# EPICS substitutions: ospreyEVRSup/Db/ospreyEVR.substitutions
#   Undefined macros
#
# P - Common record name prefix
# NAME - Device instance name

file "perEVR.template" {
pattern { P,  NAME }
  { "\$(P)", "\$(NAME)" }
}

file "perEVRhwTrigger.template" {
pattern { P,     NAME   ,  I }
  { "\$(P)", "\$(NAME)", "1" }
  { "\$(P)", "\$(NAME)", "2" }
  { "\$(P)", "\$(NAME)", "3" }
  { "\$(P)", "\$(NAME)", "4" }
}

file "perEVRevent.template" {
pattern { P,     NAME,     E }
  { "\$(P)", "\$(NAME)", "001" }
  { "\$(P)", "\$(NAME)", "002" }
  { "\$(P)", "\$(NAME)", "003" }
  { "\$(P)", "\$(NAME)", "004" }
  { "\$(P)", "\$(NAME)", "005" }
  { "\$(P)", "\$(NAME)", "006" }
  { "\$(P)", "\$(NAME)", "007" }
  { "\$(P)", "\$(NAME)", "008" }
  { "\$(P)", "\$(NAME)", "009" }
  { "\$(P)", "\$(NAME)", "010" }
  { "\$(P)", "\$(NAME)", "011" }
  { "\$(P)", "\$(NAME)", "012" }
  { "\$(P)", "\$(NAME)", "013" }
  { "\$(P)", "\$(NAME)", "014" }
  { "\$(P)", "\$(NAME)", "015" }
  { "\$(P)", "\$(NAME)", "016" }
  { "\$(P)", "\$(NAME)", "017" }
  { "\$(P)", "\$(NAME)", "018" }
  { "\$(P)", "\$(NAME)", "019" }
  { "\$(P)", "\$(NAME)", "020" }
  { "\$(P)", "\$(NAME)", "021" }
  { "\$(P)", "\$(NAME)", "022" }
  { "\$(P)", "\$(NAME)", "023" }
  { "\$(P)", "\$(NAME)", "024" }
  { "\$(P)", "\$(NAME)", "025" }
  { "\$(P)", "\$(NAME)", "026" }
  { "\$(P)", "\$(NAME)", "027" }
  { "\$(P)", "\$(NAME)", "028" }
  { "\$(P)", "\$(NAME)", "029" }
  { "\$(P)", "\$(NAME)", "030" }
  { "\$(P)", "\$(NAME)", "031" }
  { "\$(P)", "\$(NAME)", "032" }
  { "\$(P)", "\$(NAME)", "033" }
  { "\$(P)", "\$(NAME)", "034" }
  { "\$(P)", "\$(NAME)", "035" }
  { "\$(P)", "\$(NAME)", "036" }
  { "\$(P)", "\$(NAME)", "037" }
  { "\$(P)", "\$(NAME)", "038" }
  { "\$(P)", "\$(NAME)", "039" }
  { "\$(P)", "\$(NAME)", "040" }
  { "\$(P)", "\$(NAME)", "041" }
  { "\$(P)", "\$(NAME)", "042" }
  { "\$(P)", "\$(NAME)", "043" }
  { "\$(P)", "\$(NAME)", "044" }
  { "\$(P)", "\$(NAME)", "045" }
  { "\$(P)", "\$(NAME)", "046" }
  { "\$(P)", "\$(NAME)", "047" }
  { "\$(P)", "\$(NAME)", "048" }
  { "\$(P)", "\$(NAME)", "049" }
  { "\$(P)", "\$(NAME)", "050" }
  { "\$(P)", "\$(NAME)", "051" }
  { "\$(P)", "\$(NAME)", "052" }
  { "\$(P)", "\$(NAME)", "053" }
  { "\$(P)", "\$(NAME)", "054" }
  { "\$(P)", "\$(NAME)", "055" }
  { "\$(P)", "\$(NAME)", "056" }
  { "\$(P)", "\$(NAME)", "057" }
  { "\$(P)", "\$(NAME)", "058" }
  { "\$(P)", "\$(NAME)", "059" }
  { "\$(P)", "\$(NAME)", "060" }
  { "\$(P)", "\$(NAME)", "061" }
  { "\$(P)", "\$(NAME)", "062" }
  { "\$(P)", "\$(NAME)", "063" }
  { "\$(P)", "\$(NAME)", "064" }
  { "\$(P)", "\$(NAME)", "065" }
  { "\$(P)", "\$(NAME)", "066" }
  { "\$(P)", "\$(NAME)", "067" }
  { "\$(P)", "\$(NAME)", "068" }
  { "\$(P)", "\$(NAME)", "069" }
  { "\$(P)", "\$(NAME)", "070" }
  { "\$(P)", "\$(NAME)", "071" }
  { "\$(P)", "\$(NAME)", "072" }
  { "\$(P)", "\$(NAME)", "073" }
  { "\$(P)", "\$(NAME)", "074" }
  { "\$(P)", "\$(NAME)", "075" }
  { "\$(P)", "\$(NAME)", "076" }
  { "\$(P)", "\$(NAME)", "077" }
  { "\$(P)", "\$(NAME)", "078" }
  { "\$(P)", "\$(NAME)", "079" }
  { "\$(P)", "\$(NAME)", "080" }
  { "\$(P)", "\$(NAME)", "081" }
  { "\$(P)", "\$(NAME)", "082" }
  { "\$(P)", "\$(NAME)", "083" }
  { "\$(P)", "\$(NAME)", "084" }
  { "\$(P)", "\$(NAME)", "085" }
  { "\$(P)", "\$(NAME)", "086" }
  { "\$(P)", "\$(NAME)", "087" }
  { "\$(P)", "\$(NAME)", "088" }
  { "\$(P)", "\$(NAME)", "089" }
  { "\$(P)", "\$(NAME)", "090" }
  { "\$(P)", "\$(NAME)", "091" }
  { "\$(P)", "\$(NAME)", "092" }
  { "\$(P)", "\$(NAME)", "093" }
  { "\$(P)", "\$(NAME)", "094" }
  { "\$(P)", "\$(NAME)", "095" }
  { "\$(P)", "\$(NAME)", "096" }
  { "\$(P)", "\$(NAME)", "097" }
  { "\$(P)", "\$(NAME)", "098" }
  { "\$(P)", "\$(NAME)", "099" }
  { "\$(P)", "\$(NAME)", "100" }
  { "\$(P)", "\$(NAME)", "101" }
  { "\$(P)", "\$(NAME)", "102" }
  { "\$(P)", "\$(NAME)", "103" }
  { "\$(P)", "\$(NAME)", "104" }
  { "\$(P)", "\$(NAME)", "105" }
  { "\$(P)", "\$(NAME)", "106" }
  { "\$(P)", "\$(NAME)", "107" }
  { "\$(P)", "\$(NAME)", "108" }
  { "\$(P)", "\$(NAME)", "109" }
  { "\$(P)", "\$(NAME)", "110" }
  { "\$(P)", "\$(NAME)", "111" }
  { "\$(P)", "\$(NAME)", "112" }
  { "\$(P)", "\$(NAME)", "113" }
  { "\$(P)", "\$(NAME)", "114" }
  { "\$(P)", "\$(NAME)", "115" }
  { "\$(P)", "\$(NAME)", "116" }
  { "\$(P)", "\$(NAME)", "117" }
  { "\$(P)", "\$(NAME)", "118" }
  { "\$(P)", "\$(NAME)", "119" }
  { "\$(P)", "\$(NAME)", "120" }
  { "\$(P)", "\$(NAME)", "121" }
  { "\$(P)", "\$(NAME)", "122" }
  { "\$(P)", "\$(NAME)", "123" }
  { "\$(P)", "\$(NAME)", "124" }
  { "\$(P)", "\$(NAME)", "125" }
  { "\$(P)", "\$(NAME)", "126" }
  { "\$(P)", "\$(NAME)", "127" }
}
